(* IEC 61131-3 sources: Industry-PLC-LLM/data/PLCBEAD_repo/PLCBEAD_PLCEmbed-main/PLC-BEAD/Source/GEB/building_WCT, 1 file *)

(* ---- WCT.ST ---- *)
FUNCTION WCT:REAL

	VAR_INPUT
		T :	REAL;
		V :	REAL;
	END_VAR

	IF V < 5.0 OR T > 10.0 THEN
		WCT := T;
	ELSE
		WCT := 13.12 + 0.6215 * T +(0.3965 * T - 11.37) * EXP(LN(v) * 0.16);
	END_IF;

END_FUNCTION

PROGRAM program0
	VAR
		T :	REAL;
		V :	REAL;
		CEIL5_OUT : REAL;
	END_VAR

  	CEIL5_OUT := WCT(T, V);
END_PROGRAM
